TYPE FIS_VAR :
STRUCT
	CrispValue:REAL;
	Name:STRING;
	Range:ARRAY[1..2] OF REAL;
	NumberOfMF:INT;
	MF:ARRAY [1..MFmax]OF MEMBERSHIP_FUNCTION;//MF

END_STRUCT
END_TYPE

(* stored: Version 1.1.0.1, ProductVersion 3.1.4024.6
   DUT FIS_VAR: Id {ee691d09-0720-480a-8f2e-9f88962720eb} *)
